PROGRAM HydraulicPump
VAR
    
	fbHydPump: FB_HydraulicPumpControl;
	
	bMaxPressure: BOOL;
	
	fbBlink: FB_Blink_S_1;
END_VAR

fbHydPump(
	bStart         := bHydraulicUnitCmdStart,
    bStop          := bHydraulicUnitCmdStop AND NOT.bCylinderCmdDown,
    bEmergencyStop := bEStopOk,          // NC – 0=wciśnięty
    bThermalOk     := bHydraulicUnitMotorOk,        // NC – 0=zadziałany
    bPressureOk    := NOT bMaxPressure,   // czujnik NO → inwertujemy
	bOilLevel	   := TRUE,
    bEnable        := bControlOn,
	bPumpRun=> bLedHydraulicUnitOn, 
	bRunning=>.bHydraulicUintOn , 
	bFault=> , 
	bReady=> , 
	bFaultThermal=> , 
	bFaultPressure=> );
(*
Q_PumpContactor := HydPump.bPumpRun;
HMI_Alarm       := HydPump.bFault;
HMI_Ready       := HydPump.bReady;
HMI_ThermalErr  := HydPump.bFaultThermal;
HMI_PressureErr := HydPump.bFaultPressure;
*)

//=======================================================================
//			MAX. CIŚNIENIE
bMaxPressure:=Scaling.PressureAI.PV_Value>390;
//=======================================================================
//		ENABLE NA ZAWÓR PROPORCJONlNY
bProportionalValveEnable:= .bEstopOk AND (bCylinderValveUp or bCylinderValveDown);
//=======================================================================
//			LED HYDRAULIKA ZAŁACZONA
fbBlink(Tv:=T#400MS , Q=> );

IF bHydraulicUintOn THEN
 IF NOT bHydraulicUnitRunning THEN
	bLedHydraulicUnitOn:=fbBlink.Q;
	ELSIF
		 bHydraulicUnitRunning THEN
		 bLedHydraulicUnitOn:=bHydraulicUintOn;
		
	END_IF	
	ELSE
			bLedHydraulicUnitOn:=FALSE;
END_IF
//=========================================================================

END_PROGRAM

(* stored: Version 1.1.0.1, ProductVersion 3.1.4024.15
   POU HydraulicPump: Id {d8e36b58-4db9-44c2-9c45-ab5cfd7aa7ab}, SpecialFunc None *)
